// TIA Portal V20 export
VAR_GLOBAL   // PLC tag table "Unit1Em0"
   "BA010AZCRBK01.00" AT %I1000.0 : Bool;   // LEFT UNWINDER EXPEL BACKWARD
   "BA010AZCRBK01.04" AT %I1000.4 : Bool;   // LEFT TENSION CHECK SENSOR
   "BA010AZCRBK01.10" AT %I1001.0 : Bool;   // LEFT UNWINDER EXPEL FORWARD
   "BA010AZCRPM01.00" AT %Q2000.0 : Bool;   // UNWINDER LEFT AIR SHAFT ON
   "BA010AZCRSP503.00" AT %IW3100 : Int;   // LEFT UNWINDER RADIUS MEASURE
   "BA010AZCRPM05.00" AT %Q2016.0 : Bool;   // LEFT UNWINDER EXPEL FORWARD
   "BA010AZCRPM05.01" AT %Q2016.1 : Bool;   // LEFT UNWINDER EXPEL BACKWARD
END_VAR
VAR_GLOBAL CONSTANT   // user constants
   U1EM0_NO_OF_AXES : USInt := 1;   // Starts with 1. E.g., the value 4 means that 4 axes exist.
   DR1_RatedTorque : LReal := 10.6;   // UnwinderLeftAxisB
   U1EM0_JOB01 : DInt := 1;
   U1EM0_JOB02 : DInt := 2;
   U1EM0_JOB03 : DInt := 3;
   U1EM0_JOB04 : DInt := 4;
   U1EM0_JOB05 : DInt := 5;
   U1EM0_JOB06 : DInt := 6;
   U1EM0_JOB07 : DInt := 7;
   U1EM0_JOB08 : DInt := 8;
   U1EM0_JOB09 : DInt := 9;
   U1EM0_JOB10 : DInt := 10;
   U1EM0_JOB11 : DInt := 11;
   U1EM0_JOB12 : DInt := 12;
   U1EM0_JOB13 : DInt := 13;
   U1EM0_JOB14 : DInt := 14;
   U1EM0_JOB15 : DInt := 15;
   U1EM0_JOB16 : DInt := 16;
   U1EM0_JOB17 : DInt := 17;
   U1EM0_JOB18 : DInt := 18;
   U1EM0_JOB19 : DInt := 19;
   U1EM0_JOB20 : DInt := 20;
   U1EM0_JOB21 : DInt := 21;
   U1EM0_JOB22 : DInt := 22;
   U1EM0_JOB23 : DInt := 23;
   U1EM0_JOB24 : DInt := 24;
   U1EM0_JOB25 : DInt := 25;
   U1EM0_JOB26 : DInt := 26;
   U1EM0_JOB27 : DInt := 27;
   U1EM0_JOB28 : DInt := 28;
   U1EM0_JOB29 : DInt := 29;
   U1EM0_JOB30 : DInt := 30;
   U1EM0_JOB31 : DInt := 31;
   U1EM0_JOB32 : DInt := 32;
   U1EM0_JOB33 : DInt := 33;
   U1EM0_JOB34 : DInt := 34;
   U1EM0_JOB35 : DInt := 35;
   U1EM0_JOB36 : DInt := 36;
   U1EM0_JOB37 : DInt := 37;
   U1EM0_JOB38 : DInt := 38;
   U1EM0_JOB39 : DInt := 39;
   U1EM0_JOB40 : DInt := 40;
   U1EM0_JOB41 : DInt := 41;
   U1EM0_JOB42 : DInt := 42;
   U1EM0_JOB43 : DInt := 43;
   U1EM0_JOB44 : DInt := 44;
   U1EM0_JOB45 : DInt := 45;
   U1EM0_JOB46 : DInt := 46;
   U1EM0_JOB47 : DInt := 47;
   U1EM0_JOB48 : DInt := 48;
   U1EM0_JOB49 : DInt := 49;
   U1EM0_JOB50 : DInt := 50;
END_VAR
